{attribute 'GeneratedUsingTerminal: EP1816-0008-0018'}
{attribute addProperty BoxType "EP1816-0008-0018"}
{attribute addProperty Description "EP1816-0008 16 Ch. Dig. Input 24V, 10µs, D-SUB25"}
{attribute addProperty Physics "YY"}
{attribute addProperty Id "DIG_Inputs_Channel_1AT %I*DIG_Inputs_Channel_CC4551489DIG_Inputs_Channel_2AT %I*DIG_Inputs_Channel_CC4551489WcStateAT %I*WcState_9091E0EB2InfoDataAT %I*InfoData_32EB74EA10"}
{attribute addProperty CRC "1582355421"}
{attribute addProperty Size "30"}
TYPE EP1816_5E50D3DD EXTENDS EtcSlaveBoxBase_77A0E4A7 :
STRUCT
	{attribute addProperty Name "DIG_Inputs_Channel_1"}
	DIG_Inputs_Channel_1 : DIG_Inputs_Channel_CC455148;
	{attribute addProperty Name "DIG_Inputs_Channel_2"}
	DIG_Inputs_Channel_2 : DIG_Inputs_Channel_CC455148;
	{attribute addProperty Name "WcState"}
	WcState : WcState_9091E0EB;
	{attribute addProperty Name "InfoData"}
	InfoData : InfoData_32EB74EA;
END_STRUCT
END_TYPE

(* stored: Version 1.2.0.0, ProductVersion 3.1.4024.11
   DUT EP1816_5E50D3DD: Id {c6c896b0-6ac6-4ac3-a255-83d93dcffc40} *)
